{attribute 'hide_all_locals'}
FUNCTION_BLOCK INTERNAL DynamicStringBuffer
VAR_OUTPUT
	Error : Error; // Error information of this FB
END_VAR
VAR
	fifo : Tc2_Utilities.Fb_StringRingBuffer; // Necessary to buffer log data until it has been written to file.
	memory_manager : Tc3_DynamicMemory.Fb_DynMem_Manager; // Memory manager, required by DynMem_Buffer.
	dynamic_memory_buffer : Tc3_DynamicMemory.Fb_DynMem_Buffer(ipMemMan := memory_manager); // Provides dynamic buffer for Fifo. Is extended automatically if more than the
																   // default buffer size is needed.                  
	_busy : BOOL; // Buffer is busy; typically with writing data to the file system.
END_VAR

METHOD AddLine : BOOL
VAR_INPUT
	text : Tc2_System.T_MaxString; // Text to be added to the buffer
END_VAR
ResizeFifoBufferIfNecessary();
fifo.A_AddTail(putValue := Tc2_Standard.CONCAT(Tc2_Standard.LEFT(text, 254), '$N'));
END_METHOD

METHOD AddString : BOOL
VAR_INPUT
	text : Tc2_System.T_MaxString; // String to be added to the buffer
END_VAR
ResizeFifoBufferIfNecessary();
fifo.A_AddTail(putValue := text);
END_METHOD

METHOD PRIVATE AllocateBuffer : BOOL // Allocates buffer FOR the fifo.
VAR_INPUT
	bufferSize : UDINT; // Initial buffer size in BYTEs for fifo buffer.
END_VAR
dynamic_memory_buffer.CreateBuffer(nSize:=bufferSize, bReset:=TRUE);
fifo.pBuffer := dynamic_memory_buffer.pBuffer;
fifo.cbBuffer := bufferSize;
END_METHOD

{attribute 'monitoring':='call'}
PROPERTY PUBLIC Busy : BOOL
GET // PUBLIC
Busy := _busy;
END_GET
SET // PRIVATE
_busy := Busy;
END_SET
END_PROPERTY

METHOD FB_exit : BOOL
VAR_INPUT
	bInCopyCode : BOOL; // if TRUE, the exit method is called for exiting an instance that is copied afterwards (online change).
END_VAR
dynamic_memory_buffer.Clear();
END_METHOD

METHOD FlushCache : BOOL
fifo.A_Reset();
END_METHOD

METHOD INTERNAL Init : BOOL
VAR_INPUT
	bufferSize : UDINT; // Initial buffer size in BYTEs for fifo buffer.
END_VAR
AllocateBuffer(bufferSize);
END_METHOD

{attribute 'hide_all_locals'}
METHOD PersistToFile : BOOL
VAR_INPUT
	enable: BOOL; // TRUE starts persistence mechanism
	fileName : Tc2_System.T_MaxString; // File name including its path
END_VAR
VAR_INST
	state : PersistToFileState;
	
	file_open : Tc2_System.FB_FileOpen;
	file_handle : UINT;
	
	file_write : Tc2_System.FB_FileWrite;
	lockFileWriteToForceRisingEdge : BOOL; // filePuts can only be executed every other cycle
										 // since it needs a rising edge to execute.
	file_close : Tc2_System.FB_FileClose;
	
	buffer : ARRAY[0..Constants.BufferSize] OF BYTE;
	currentBufferPos : UDINT;
	fifo_head_string : Tc2_System.T_MaxString;
	fifo_head_length : UDINT;
	fifo_head_bytes : ARRAY[0..Tc2_System.Max_String_Length] OF BYTE;
	i : UINT;
END_VAR
VAR CONSTANT
	NetId : STRING := '';
	Timeout : TIME := Tc2_System.Default_Ads_Timeout;
	MaxLogsPerCycle : UINT := UDINT_TO_UINT(Constants.BufferSize / Tc2_System.Max_String_Length);
	MaxBufferPosition : UDINT := SIZEOF(buffer) - Tc2_System.Max_String_Length;
END_VAR
// State machine
// Using if-statements instead of case for performance reasons:
// Some states execute instantly and allow thus the next state 
// to start within the same plc cycle.

// *** I D L E ***
IF state = PersistToFileState.Idle THEN
	lockFileWriteToForceRisingEdge := FALSE;
	IF fifo.nCount > 0 AND enable THEN 
		lockFileWriteToForceRisingEdge := FALSE;
		state := PersistToFileState.OpenFile;
	END_IF
END_IF
    
// *** O P E N   F I L E ***
file_open(
	sNetId := NetId,
	sPathName := fileName,
	nMode := Tc2_System.Fopen_ModeAppend OR Tc2_System.Fopen_ModeText, 
	ePath := Tc2_System.Path_Generic,
	bExecute := (state = PersistToFileState.OpenFile),
	tTimeout := Timeout,
	hFile => file_handle
);

IF state = PersistToFileState.OpenFile THEN
	IF file_open.bError THEN
		state := PersistToFileState.CloseFile;
	ELSIF NOT file_open.bBusy THEN
		state := PersistToFileState.GetStringFromFifo; 
	END_IF
END_IF 

// *** P O P   F R O M   F I F O ***
IF state = PersistToFileState.GetStringFromFifo THEN
	IF NOT lockFileWriteToForceRisingEdge THEN
		currentBufferPos := 0;
		FOR i:=0 TO MaxLogsPerCycle DO
			IF fifo.nCount <= 0 THEN EXIT; END_IF
			IF currentBufferPos >= MaxBufferPosition THEN EXIT; END_IF
			
			fifo.A_RemoveHead(getValue => fifo_head_string); 
			fifo_head_bytes := Tc2_Utilities.MaxString_To_ByteArr(fifo_head_string);
			fifo_head_length := INT_TO_UDINT(Tc2_System.Len(fifo_head_string));
			Tc2_System.MemCpy(
				destAddr := ADR(buffer) + SIZEOF(BYTE) * currentBufferPos,
				srcAddr := ADR(fifo_head_bytes),
				n := fifo_head_length
			);    
			currentBufferPos := currentBufferPos + fifo_head_length;  
		END_FOR
		state := PersistToFileState.AppendDataToFile;
	END_IF
	lockFileWriteToForceRisingEdge := FALSE;
END_IF
  
// *** W R I T E   T O   F I L E ***
file_write(
	sNetId := NetId, 
	hFile := file_handle, 
	pWriteBuff := ADR(buffer),
	cbWriteLen := currentBufferPos,
	bExecute := state = PersistToFileState.AppendDataToFile, 
	tTimeout := Timeout
); 

IF state = PersistToFileState.AppendDataToFile THEN
	lockFileWriteToForceRisingEdge := TRUE;   
	IF file_write.bError THEN
		state := PersistToFileState.CloseFile;
	ELSIF fifo.nCount > 0 AND NOT file_write.bBusy THEN
		state := PersistToFileState.GetStringFromFifo; 
	ELSIF fifo.nCount = 0 THEN
		state := PersistToFileState.CloseFile;
	END_IF
END_IF
    
// *** C L O S E   F I L E ***
file_close(
	sNetId := NetId,
	hFile := file_handle, 
	bExecute := (state = PersistToFileState.CloseFile),
	tTimeout := Timeout
);

IF state = PersistToFileState.CloseFile THEN
	IF NOT file_close.bBusy THEN
		state := PersistToFileState.Idle;
	END_IF
END_IF

// Close file in case of error
IF file_open.bError THEN
	state := PersistToFileState.CloseFile;
END_IF

IF file_write.bError THEN
	state := PersistToFileState.CloseFile;
END_IF

IF NOT fifo.bOk
	AND fifo.nCount > 0
	AND state <> PersistToFileState.Idle
THEN 
  state := PersistToFileState.CloseFile; 
END_IF

// Error handling
IF file_open.bError THEN
  Error.Active := TRUE;
  Error.Code := ErrorCodes.OpeningFileFailed;
  Error.Info := Tc2_Standard.ConCat('Opening file failed. Error thrown by FB_FileOpen. Consult Beckhoff InfoSys. Internal Error: ', UDINT_TO_STRING(file_open.nErrId));
ELSIF file_write.bError THEN
  Error.Active := TRUE;
  Error.Code := ErrorCodes.WritingToFileFailed;
  Error.Info := Tc2_Standard.ConCat('Writing to file failed. Error thrown by FB_FileWrite. Consult Beckhoff InfoSys. Internal Error: ', UDINT_TO_STRING(file_write.nErrId));
ELSIF file_close.bError THEN
  Error.Active := TRUE;
  Error.Code := ErrorCodes.ClosingFileFailed;
  Error.Info := Tc2_Standard.ConCat('Closing file failed. Error thrown by FB_FileClose. Consult Beckhoff InfoSys. Internal Error: ', UDINT_TO_STRING(file_close.nErrId));
ELSIF NOT fifo.bOk AND fifo.nCount > 0 THEN
  Error.Active := TRUE;
  Error.Code := ErrorCodes.FifoOverflow;
  Error.Info := 'FIFO overflow. Check if plc has enough free memory.';
ELSE
  Error.Active := FALSE;
  Error.Code := ErrorCodes.None;
  Error.Info := '';
END_IF

// Set busy state
Busy := (state <> PersistToFileState.Idle OR fifo.nCount > 0);

(* Uncomment for cyclic logging of state machine, buffer usage & errors

ADSLOGSTR(ADSLOG_MSGTYPE_LOG, 
  Tc2_Standard.CONCAT('****DynamicStringBuffer.state:', 
  Tc2_Standard.CONCAT(UINT_TO_STRING(state),
  Tc2_Standard.CONCAT(', DynamicStringBuffer.hFile:', UINT_TO_STRING(hFile)))), '');

ADSLOGSTR(ADSLOG_MSGTYPE_LOG, 
  Tc2_Standard.CONCAT('****Fifo: used ', 
  Tc2_Standard.CONCAT(UDINT_TO_STRING(Fifo.cbSize),
  Tc2_Standard.CONCAT(' of ', UDINT_TO_STRING(Fifo.cbBuffer)))), '');
  
IF Error.Active THEN
  ADSLOGSTR(ADSLOG_MSGTYPE_LOG, 
    Tc2_Standard.CONCAT('****DynamicStringBuffer.Error: ', Error.Info), 
    '');  
END_IF
*)
END_METHOD

METHOD PopHead : Tc2_System.T_MaxString
VAR_INST
	headString : Tc2_System.T_MaxString;
END_VAR
fifo.A_RemoveHead(getValue => headString);
PopHead := headString;
END_METHOD

// Resizes the buffer for the FIFO if necessary
METHOD PRIVATE ResizeFifoBufferIfNecessary : BOOL
VAR
	requiredSize : UDINT;
	newSize : DINT;
END_VAR
requiredSize := fifo.cbSize + (Tc2_System.MAX_STRING_LENGTH + Constants.FifoOverhead);

IF requiredSize > fifo.cbBuffer THEN
	dynamic_memory_buffer.Resize(nSize := requiredSize*SIZEOF(BYTE), bPreserve:=TRUE, bReset:=TRUE);
	fifo.pBuffer := dynamic_memory_buffer.pBuffer;
	fifo.cbBuffer := requiredSize;
END_IF
END_METHOD

END_FUNCTION_BLOCK

(* stored: Version 1.1.0.1
   POU DynamicStringBuffer: Id {21d3978e-ed2d-4d88-a5a3-251abdab9bf2}, SpecialFunc None
   Method AddLine: Id {ce3ec4cc-b756-4933-9bf5-8c247928a37b}
   Method AddString: Id {a0f9e6c7-f718-4422-bda0-36c1c9bb9e51}
   Method AllocateBuffer: Id {98da2d6e-0ea8-40ce-b189-8716915313b6}
   Property Busy: Id {2d59c975-f5f3-43ee-b807-9921c8621e41}
   Get Get: Id {457d8bae-62af-4662-8fbf-083e3b64cbd5}
   Set Set: Id {32dc2e66-ed23-41fe-ac22-23e12a7e5bd2}
   Method FB_exit: Id {a148b568-f2ae-4b33-a578-b07871ea4591}
   Method FlushCache: Id {9c6f1b89-2ada-484b-9016-16e31ae2692c}
   Method Init: Id {48a87aab-d8d7-4f6e-a893-ab8947874696}
   Method PersistToFile: Id {9ee7c4b9-2795-4bc0-891b-4613f9526c2b}
   Method PopHead: Id {1a26e5cc-ccfe-473c-968b-3f3e15197a61}
   Method ResizeFifoBufferIfNecessary: Id {c0f238dc-776d-4004-a550-6fb58f5b5a2e} *)
